FUNCTION_BLOCK FB_Blinking
VAR_IN_OUT
	io_xBlinking		: BOOL;
END_VAR
VAR
	tBlink     		: TON;       
    xBlink     		: BOOL;    
END_VAR

tBlink(IN := TRUE, PT := T#500MS);  

IF tBlink.Q THEN
    xBlink := NOT xBlink;     
    tBlink(IN := FALSE);        
ELSE
    tBlink(IN := TRUE);       
END_IF

io_xBlinking := xBlink;

END_FUNCTION_BLOCK

(* stored: Version 1.1.0.1
   POU FB_Blinking: Id {125c5226-143d-4d56-a3ad-946889c8f97e}, SpecialFunc None *)
